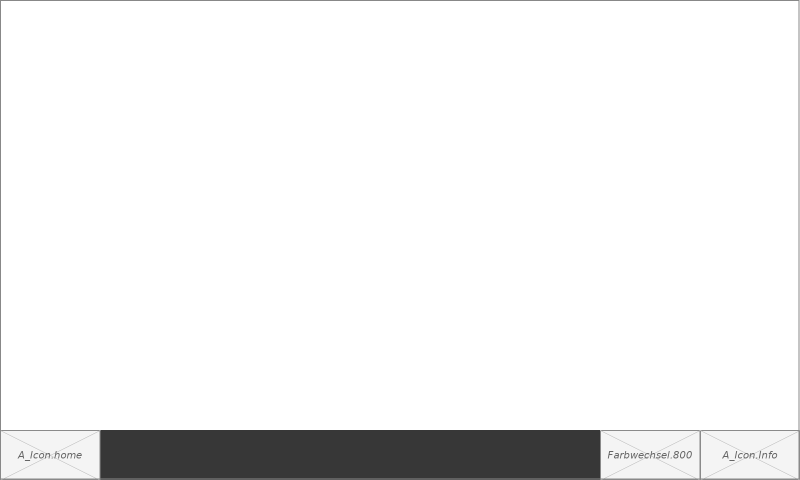
VISUALIZATION Fusszeile  // 800x480
    Rectangle (0,430 800x50)
    Image (600,430 100x50), image: Farbwechsel.800
        p84334746: Visu.s_Status_AL_Button
        OnMouseClick: change screen: Alarmliste
    Image (700,430 100x50), image: A_Icon.Info
    Image (0,430 100x50), image: A_Icon.home
        OnMouseClick: change screen: Home
END_VISUALIZATION

(* stored: Version 1.1.0.1, ProductVersion 3.1.4022.6
   Visu Fusszeile: Id {a02a0b92-f3ed-4627-8b71-b92128410167} *)
